{attribute 'qualified_only'}
VAR_GLOBAL
	PR1 AT %Q*: BOOL;	// Parkplätze Reihe 1
	PR2 AT %Q*: BOOL;	// Parkplätze Reihe 2
	PR3 AT %Q*: BOOL;	// Parkplätze Reihe 3
	PR4 AT %Q*: BOOL;	// Parkplätze Reihe 4
END_VAR

(* stored: Version 1.1.0.1, ProductVersion 3.1.4024.4
   GVL SimDA: Id {efa3d63a-96e1-4204-b1e7-9f3703bd4f03} *)
